TYPE "ValveSts"
VERSION : 0.1
// Block: ValveSts
   STRUCT
      AlarmPresence : Bool;
      RestPermit : Bool;
      RestInProgress : Bool;
      IsAtRest : Bool;
      WorkPermit : Bool;
      WorkInProgress : Bool;
      IsAtWork : Bool;
      StandStill : Bool;
   END_STRUCT;

END_TYPE
